# B&R Automation Studio project ChoiceBagging_SSBP
Automation Studio 4.5.2.102; Single Spout Bag Placer; technology packages: mapp 5.6.0

## Configuration SSBP1

CPU X20CP0410, AutomationRuntime D4.52, Build 4.1.2, Vc V4.52.0

### Hardware
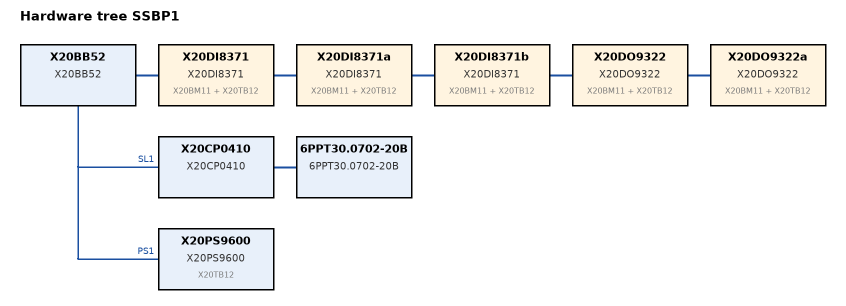
```
6PPT30.0702-20B : 6PPT30.0702-20B v1.1.0.0  [ETH1 -> X20CP0410.IF2 [Cable Type=PowerlinkCable, Length=10, Version=1.0.0.2]]
  Terminal = true
  PasswordVNC = 
  PasswordCIFS = 
  PasswordService = 
  VncKeyMappingFile = VC\6PPT30.0702-20B.dis
  VncRefreshRate = 400
X20BB52 : X20BB52 v1.1.0.0
X20BM11 : X20BM11 v1.0.0.1  [X2X1 -> X20BB52.IF6]
X20BM11a : X20BM11 v1.0.0.1  [X2X1 -> X20BM11d.X2X2]
X20BM11b : X20BM11 v1.0.0.1  [X2X1 -> X20BM11.X2X2]
X20BM11c : X20BM11 v1.0.0.1  [X2X1 -> X20BM11a.X2X2]
X20BM11d : X20BM11 v1.0.0.1  [X2X1 -> X20BM11b.X2X2]
X20CP0410 : X20CP0410 v1.2.1.0  [SL -> X20BB52.SL1]
  Connector IF2:
    ActivateDevice = 1
    Mode = Manual
    InternetAddress = 10.128.131.200
    SubnetMask = 255.255.255.0
    InaNodeNumber = 0
    Vnc1
    VncVcObjectName1 = Visu
    VncKeyMappingFile1 = VC\PS2-Keyboard.dis
    VncRefreshRate1 = 250
  ConfigurationID = ChoiceBagging_SSBP_SSBP1
  EnableUsbRemoteInstall = 1
  TimerDeviceType = SWIOTIMER
  Cyclic1Duration = 10000
  Cyclic1Tolerance = 10000
  Cyclic1Output = 1
  Cyclic2Duration = 20000
  Cyclic2Tolerance = 20000
  Cyclic3Duration = 50000
  Cyclic3Tolerance = 50000
  Cyclic4Duration = 100000
  Cyclic4Tolerance = 100000
  Cyclic5Duration = 200000
  Cyclic5Tolerance = 200000
  Cyclic6Duration = 500000
  Cyclic6Tolerance = 500000
  Cyclic7Duration = 1000000
  Cyclic7Tolerance = 1000000
  Cyclic8Duration = 10000
  Cyclic8Tolerance = 30000000
  ActivateOpcUa = 1
  OpcUaInformationModels_PV_Version = 1
X20DI8371 : X20DI8371 v1.0.2.0  [SS1 -> X20TB12a.SS; SL -> X20BM11.SL1]
  Supervision = off
X20DI8371a : X20DI8371 v1.0.2.0  [SS1 -> X20TB12c.SS; SL -> X20BM11b.SL1]
  Supervision = off
X20DI8371b : X20DI8371 v1.0.2.0  [SS1 -> X20TB12e.SS; SL -> X20BM11d.SL1]
X20DO9322 : X20DO9322 v1.0.3.0  [SS1 -> X20TB12b.SS; SL -> X20BM11a.SL1]
  Supervision = off
X20DO9322a : X20DO9322 v1.0.3.0  [SS1 -> X20TB12d.SS; SL -> X20BM11c.SL1]
  Supervision = off
X20PS9600 : X20PS9600 v1.0.1.0  [PS -> X20BB52.PS1; SS1 -> X20TB12.SS]
  Supervision = off
X20TB12 : X20TB12 v1.0.0.0
X20TB12a : X20TB12 v1.0.0.0
X20TB12b : X20TB12 v1.0.0.0
X20TB12c : X20TB12 v1.0.0.0
X20TB12d : X20TB12 v1.0.0.0
X20TB12e : X20TB12 v1.0.0.0
```

### IoMap.iom - X20CP0410/IoMap.iom
```iecst
VAR_CONFIG
	::gModuleOK.PowerSupply AT %IX."X20PS9600".ModuleOk;
	::gModuleOK.DigitalInput AT %IX."X20DI8371".ModuleOk;
	::gModuleOK.DigitalOutput AT %IX."X20DO9322".ModuleOk;
	::gModuleOK.DigitalInputa AT %IX."X20DI8371a".ModuleOk;
	::gModuleOK.DigitalOutputa AT %IX."X20DO9322a".ModuleOk;
	::gdi.L1CarriageRight AT %IX."X20DI8371".DigitalInput01;
	::gdi.L2CarriageLeft AT %IX."X20DI8371".DigitalInput02;
	::gdi.L3BagLifterUpper AT %IX."X20DI8371".DigitalInput03;
	::gdi.L4BagLifterLower AT %IX."X20DI8371".DigitalInput04;
	::gdi.L5DuckBillLeft AT %IX."X20DI8371".DigitalInput05;
	::gdi.L6DuckBillRight AT %IX."X20DI8371".DigitalInput06;
	::gdi.L7GripperOpen AT %IX."X20DI8371".DigitalInput07;
	::gdi.L8VacuumConfirm AT %IX."X20DI8371".DigitalInput08;
	::gdi.L9SwingArmUpper AT %IX."X20DI8371a".DigitalInput01;
	::gdi.L10SwingArmLower AT %IX."X20DI8371a".DigitalInput02;
	::gdi.L11EmptyBagInboundConv AT %IX."X20DI8371a".DigitalInput03;
	::gdi.L12Cyl7SpreaderSwitch AT %IX."X20DI8371a".DigitalInput04;
	::gdi.Bagger1Ready AT %IX."X20DI8371a".DigitalInput05;
	::gdi.Bagger2OnSpout AT %IX."X20DI8371a".DigitalInput06;
	::gdi.ConveyorOn AT %IX."X20DI8371a".DigitalInput07;
	::gdo.Cyl1CarriageLeft AT %QX."X20DO9322".DigitalOutput01;
	::gdo.Cyl1CarriageRight AT %QX."X20DO9322".DigitalOutput02;
	::gdo.Cyl2SwingArmUp AT %QX."X20DO9322".DigitalOutput03;
	::gdo.Cyl2SwingArmDown AT %QX."X20DO9322".DigitalOutput04;
	::gdo.Cyl3EmptyBagUp AT %QX."X20DO9322".DigitalOutput05;
	::gdo.Cyl3DownToEmptyBag AT %QX."X20DO9322".DigitalOutput06;
	::gdo.Cyl4DuckBillLeft AT %QX."X20DO9322".DigitalOutput07;
	::gdo.Cyl4DuckBillRight AT %QX."X20DO9322".DigitalOutput08;
	::gdo.Cyl5DuckBillIn AT %QX."X20DO9322".DigitalOutput09;
	::gdo.Cyl5DuckBillOut AT %QX."X20DO9322".DigitalOutput10;
	::gdo.Cyl6DuckBillOpen AT %QX."X20DO9322".DigitalOutput11;
	::gdo.Cyl6DuckBillClose AT %QX."X20DO9322".DigitalOutput12;
	::gdo.Cyl7Spreader AT %QX."X20DO9322a".DigitalOutput01;
	::gdo.Cyl8DropOpen AT %QX."X20DO9322a".DigitalOutput02;
	::gdo.Cyl8GripClose AT %QX."X20DO9322a".DigitalOutput03;
	::gdo.Vac1 AT %QX."X20DO9322a".DigitalOutput04;
	::gdo.Purge1 AT %QX."X20DO9322a".DigitalOutput05;
	::gdi.SafeToRun AT %IX."X20DI8371a".DigitalInput08;
	::gdi.ChairDischarge AT %IX."X20DI8371b".DigitalInput01;
	::gModuleOK.DigitalInputb AT %IX."X20DI8371b".ModuleOk;
	::gdo.Alarm AT %QX."X20DO9322a".DigitalOutput06;
	::gdo.Running AT %QX."X20DO9322a".DigitalOutput07;
	::gdi.SealerArmUp AT %IX."X20DI8371b".DigitalInput02;
	::gdi.ChairIn AT %IX."X20DI8371b".DigitalInput03;
END_VAR
```

### Config.mpalarmxcore - X20CP0410/mappServices/Config.mpalarmxcore
```
Element gAlarmXCore (Type=mpalarmxcore)
  mapp.AlarmX.Core.Configuration:
    [0]:
      Name = HomingTimeout
      Message = Timeout while homing machine.
      Code = 1
    [1]:
      Name = SafetyStatus
      Message = Safety status error not OK.
      Code = 2
    [2]:
      Name = ConveyorStatus
      Message = Conveyor status error not OK.
      Code = 3
    [3]:
      Name = ModuleStatus
      Message = Hardware module not OK.
      Code = 4
    [4]:
      Name = VacuumFailure
      Message = Vacuum confirmation failure.
      Code = 5
    [5]:
      Name = Bagger2Failure
      Message = No bag on spout.
      Code = 6
```

## Logical view

Binary libraries used (declarations not repeated): operator, runtime, astime, AsIecCon, AsArSdm, brsystem, MpBase, standard, sys_lib, MpAlarmX 5.06.0

### Global.typ - Global data types
```iecst
TYPE
	MachineState_type : 	STRUCT  (*State machine*)
		Sub0 : BOOL; (*Subroutine 0*)
		Sub1 : BOOL; (*Subroutine 1*)
		Sub2 : BOOL; (*Subroutine 2*)
		Sub3 : BOOL; (*Subroutine 3*)
		Sub4 : BOOL; (*Subroutine 4*)
		Sub5 : BOOL; (*Subroutine 5*)
		Sub6 : BOOL; (*Subroutine 6*)
		Sub7 : BOOL; (*Subroutine 7*)
		Sub8 : BOOL; (*Subroutine 8*)
		Sub9 : BOOL; (*Subroutine 9*)
	END_STRUCT;
	di_type : 	STRUCT  (*Digital inputs*)
		L1CarriageRight : BOOL; (*Carriage limit right*)
		L2CarriageLeft : BOOL; (*Carriage limit left*)
		L3BagLifterUpper : BOOL; (*Bag lifter limit upper*)
		L4BagLifterLower : BOOL; (*Bag lifter limit lower*)
		L5DuckBillLeft : BOOL; (*Duck bill limit left*)
		L6DuckBillRight : BOOL; (*Duck bill limit right*)
		L7GripperOpen : BOOL; (*Gripper open limit*)
		L8VacuumConfirm : BOOL; (*Vacuum confirmation*)
		L9SwingArmUpper : BOOL; (*Swing arm limit upper*)
		L10SwingArmLower : BOOL; (*Swing arm limit lower*)
		L11EmptyBagInboundConv : BOOL; (*Empty bag inbound conveyor*)
		L12Cyl7SpreaderSwitch : BOOL; (*Activate Cyl7 switch*)
		Bagger1Ready : BOOL; (*Ready signal from bagger*)
		Bagger2OnSpout : BOOL; (*No bag on spout from bagger*)
		ConveyorOn : BOOL; (*Conveyor on signal from robotic palletizer*)
		SafeToRun : BOOL; (*Safe to run signal from safety light curtain*)
		ChairDischarge : BOOL; (*Chair discharge signal*)
		SealerArmUp : BOOL; (*Sealer arm up signal*)
		ChairIn : BOOL; (*Chair in signal*)
	END_STRUCT;
	do_type : 	STRUCT  (*Digital outputs*)
		Cyl1CarriageLeft : BOOL; (*Move carriage left*)
		Cyl1CarriageRight : BOOL; (*Move carriage right*)
		Cyl2SwingArmUp : BOOL; (*Move swinging arm up*)
		Cyl2SwingArmDown : BOOL; (*Move swinging arm down*)
		Cyl3EmptyBagUp : BOOL; (*Lift empty bags up*)
		Cyl3DownToEmptyBag : BOOL; (*Move down to empty bags*)
		Cyl4DuckBillLeft : BOOL; (*Move duck bill assembly left*)
		Cyl4DuckBillRight : BOOL; (*Move duck bill assembly right*)
		Cyl5DuckBillIn : BOOL; (*Move duck bill in*)
		Cyl5DuckBillOut : BOOL; (*Move duck bill out*)
		Cyl6DuckBillOpen : BOOL; (*Open duck bill*)
		Cyl6DuckBillClose : BOOL; (*Close duck bill*)
		Cyl7Spreader : BOOL; (*Bag valve spreader*)
		Cyl8DropOpen : BOOL; (*Drop bag*)
		Cyl8GripClose : BOOL; (*Grip bag*)
		Vac1 : BOOL; (*Attach bag to bag lifter*)
		Purge1 : BOOL; (*Purge vacuum lines*)
		Alarm : BOOL; (*Error present*)
		Running : BOOL; (*Machine running*)
	END_STRUCT;
	ModuleOK_type : 	STRUCT  (*Module statuses*)
		PowerSupply : BOOL; (*X20PS9600 status*)
		DigitalInput : BOOL; (*X20DI8371 status*)
		DigitalOutput : BOOL; (*X20DO9322 status*)
		DigitalInputa : BOOL; (*X20DI8371a status*)
		DigitalOutputa : BOOL; (*X20DO9322a status*)
		DigitalInputb : BOOL; (*X20DI8371b status*)
	END_STRUCT;
	Timer_type : 	STRUCT  (*System timers*)
		HomePos : TIME; (*Homing Position timer value*)
		BagOnSpout : TIME; (*Bag on Spout timer value*)
		VacuumConfirm : TIME; (*Vacuum Confirmation timer value*)
		Cyl5 : TIME; (*Cyl 5 timer value*)
		Cyl6 : TIME; (*Cyl 6 timer value*)
		Cyl7 : TIME; (*Cyl 7 timer value*)
		GripperRetract : TIME; (*Gripper retract timer value*)
		SwingArm : TIME; (*Swing arm timer value*)
	END_STRUCT;
	Machine_type : 	STRUCT  (*Machine structure type*)
		Cmd : MachineCmd_type; (*Machine commands*)
		Par : MachinePar_type; (*Machine parameters*)
		Sts : MachineSts_type; (*Machine statuses*)
	END_STRUCT;
	MachineCmd_type : 	STRUCT  (*Machine commands*)
		Home : BOOL; (*Home*)
		Initialize : BOOL; (*Initialize - start from home*)
		Start : BOOL; (*Start machine*)
		Stop : BOOL; (*Stop machine*)
		ErrorReset : BOOL; (*Reset error*)
		Wait : BOOL; (*Wait state*)
		Pause : BOOL; (*Pause machine*)
		Resume : BOOL; (*Resume subroutine*)
	END_STRUCT;
	MachinePar_type : 	STRUCT  (*Machine parameters*)
		VacuumFail : UDINT; (*Vacuum confirmation failure*)
		VacuumFailTotal : UDINT; (*Vacuum confirmation failure total*)
		Bagger2Fail : UDINT; (*Bagger 2 on Spout failure*)
		Bagger2FailTotal : UDINT; (*Bagger 2 on Spout failure total*)
	END_STRUCT;
	MachineSts_type : 	STRUCT  (*Machine statuses*)
		IsHomed : BOOL; (*Is homed*)
		Cyl6LimitClose : BOOL; (*Cyl 6 timer feedback - duck bill close*)
		Cyl6LimitOpen : BOOL; (*Cyl 6 timer feedback - duck bill open*)
		Cyl5LimitOut : BOOL; (*Cyl 5 timer feedback - duck bill out*)
		Cyl5LimitIn : BOOL; (*Cyl 5 timer feedback - duck bill in*)
		Error : BOOL; (*Error detected*)
		HomePosTimeout : BOOL; (*Home Position timeout*)
		VacuumTimeout : BOOL; (*Vacuum Confirmation timeout*)
		AttemptsLeft : BOOL; (*Attempts left before error - vacuum*)
		NoAttemptsLeft : BOOL; (*No vacuum attempts left - error*)
		Bagger2Timeout : BOOL; (*Bag on Spout timeout*)
		BaggerAttemptsLeft : BOOL; (*Attempts left before error - Bagger 2*)
		NoBaggerAttemptsLeft : BOOL; (*No Bagger 2 attempts left - error*)
	END_STRUCT;
	Input_type : 	STRUCT  (*Machine inputs*)
		L1CarriageRight : BOOL; (*Carriage limit right*)
		L2CarriageLeft : BOOL; (*Carriage limit left*)
		L3BagLifterUpper : BOOL; (*Bag lifter limit upper*)
		L4BagLifterLower : BOOL; (*Bag lifter limit lower*)
		L5DuckBillLeft : BOOL; (*Duck bill limit left*)
		L6DuckBillRight : BOOL; (*Duck bill limit right*)
		L7GripperOpen : BOOL; (*Gripper open limit*)
		L8VacuumConfirm : BOOL; (*Vacuum confirmation*)
		L9SwingArmUpper : BOOL; (*Swing arm limit upper*)
		L10SwingArmLower : BOOL; (*Swing arm limit lower*)
		L11EmptyBagInboundConv : BOOL; (*Empty bag inbound conveyor*)
		L12Cyl7SpreaderSwitch : BOOL; (*Activate Cyl7 switch*)
		Bagger1Ready : BOOL; (*Ready signal from bagger*)
		Bagger2OnSpout : BOOL; (*No bag on spout from bagger*)
		ConveyorOn : BOOL; (*Conveyor on signal from robotic palletizer*)
		SafeToRun : BOOL; (*Safe to run signal from safety light curtain*)
		ChairDischarge : BOOL; (*Chair discharge signal*)
		SealerArmUp : BOOL; (*Sealer arm up signal*)
		ChairIn : BOOL; (*Chair in signal*)
	END_STRUCT;
	Output_type : 	STRUCT  (*Machine outputs*)
		Cyl1CarriageLeft : BOOL; (*Move carriage left*)
		Cyl1CarriageRight : BOOL; (*Move carriage right*)
		Cyl2SwingArmUp : BOOL; (*Move swinging arm up*)
		Cyl2SwingArmDown : BOOL; (*Move swinging arm down*)
		Cyl3EmptyBagUp : BOOL; (*Lift empty bags up*)
		Cyl3DownToEmptyBag : BOOL; (*Move down to empty bags*)
		Cyl4DuckBillLeft : BOOL; (*Move duck bill assembly left*)
		Cyl4DuckBillRight : BOOL; (*Move duck bill assembly right*)
		Cyl5DuckBillIn : BOOL; (*Move duck bill in*)
		Cyl5DuckBillOut : BOOL; (*Move duck bill out*)
		Cyl6DuckBillOpen : BOOL; (*Open duck bill*)
		Cyl6DuckBillClose : BOOL; (*Close duck bill*)
		Cyl7Spreader : BOOL; (*Bag valve spreader*)
		Cyl8DropOpen : BOOL; (*Drop bag*)
		Cyl8GripClose : BOOL; (*Grip bag*)
		Vac1 : BOOL; (*Attach bag to bag lifter*)
		Purge1 : BOOL; (*Purge vacuum lines*)
		Alarm : BOOL; (*Error detected*)
		Running : BOOL; (*Machine Running*)
	END_STRUCT;
	ErrorID_enum :
		( (*Error ID enumeration*)
		HOMING_TIMEOUT := 1, (*Homing position timeout*)
		SAFE_TO_RUN := 2, (*Machine not Safe to Run*)
		CONVEYOR := 3, (*Conveyor not on*)
		MODULE_OK := 4, (*Module OK status error*)
		VACUUM_FAILURE := 5, (*Vacuum failure (after 3 attempts)*)
		BAG_ON_SPOUT_FAILURE := 6 (*No Bag on spout (after 3 attempts)*)
		);
END_TYPE
```

### Global.var - Global variables
```iecst
VAR
	gdi : di_type; (*Digital inputs*)
	gdo : do_type; (*Digital outputs*)
	gModuleOK : ModuleOK_type; (*Module statuses*)
	gTimer : Timer_type; (*System timers*)
	gErrorID : UDINT; (*Error ID*)
	gMachine : Machine_type; (*Machine process variable*)
	gInput : Input_type; (*Machine inputs process variable*)
	gOutput : Output_type; (*Machine outputs process variable*)
	gMachineState : MachineState_type; (*State machine process variable*)
END_VAR
```


### Program Logical/MainCtrl (IEC)

#### Cyclic.ld - Cyclic code
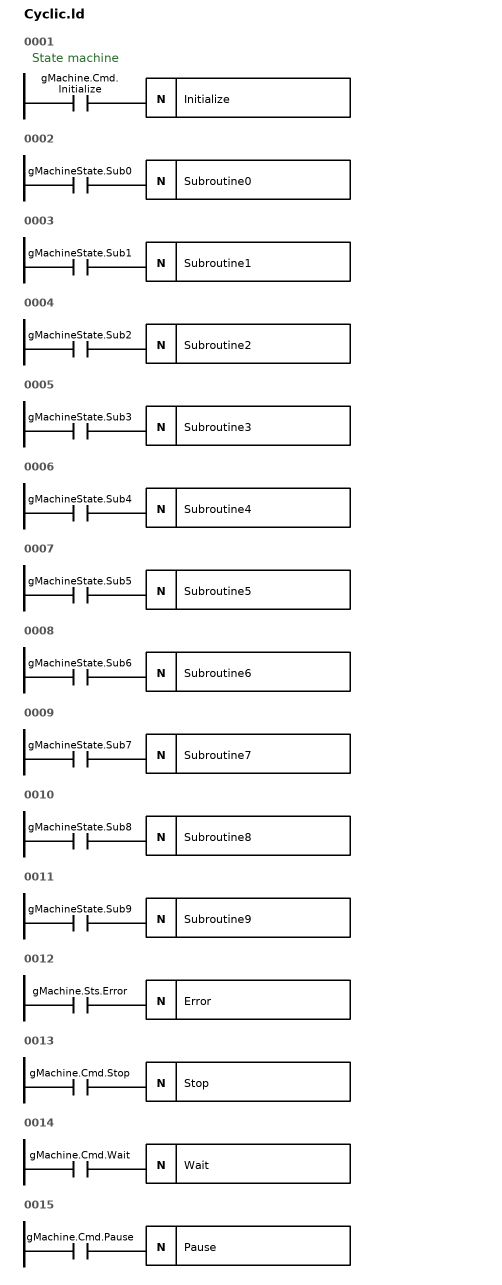
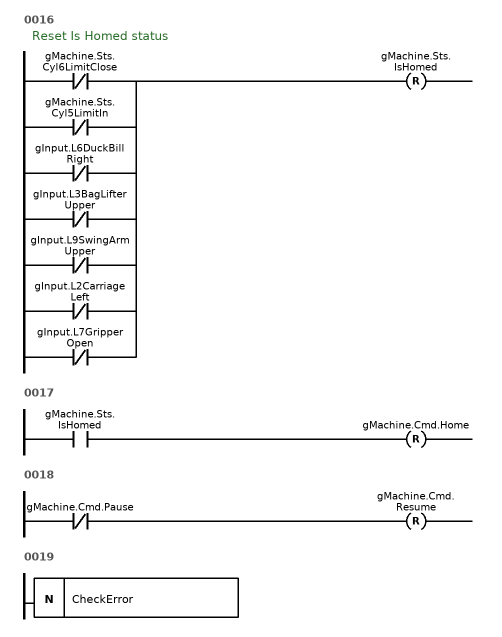
Ladder, written as Structured Text:
```iecst
(*********************************************************************************
 * Copyright: 	Hartfiel Automation
 * Author:    	cashley
 * Created:   	August 5, 2019/2:01 PM
 * Description: This file contains the main control logic for the machine.
 *********************************************************************************)
 PROGRAM _CYCLIC
(* Network 1: State machine *)
IF gMachine.Cmd.Initialize THEN Initialize; END_IF;

(* Network 2 *)
IF gMachineState.Sub0 THEN Subroutine0; END_IF;

(* Network 3 *)
IF gMachineState.Sub1 THEN Subroutine1; END_IF;

(* Network 4 *)
IF gMachineState.Sub2 THEN Subroutine2; END_IF;

(* Network 5 *)
IF gMachineState.Sub3 THEN Subroutine3; END_IF;

(* Network 6 *)
IF gMachineState.Sub4 THEN Subroutine4; END_IF;

(* Network 7 *)
IF gMachineState.Sub5 THEN Subroutine5; END_IF;

(* Network 8 *)
IF gMachineState.Sub6 THEN Subroutine6; END_IF;

(* Network 9 *)
IF gMachineState.Sub7 THEN Subroutine7; END_IF;

(* Network 10 *)
IF gMachineState.Sub8 THEN Subroutine8; END_IF;

(* Network 11 *)
IF gMachineState.Sub9 THEN Subroutine9; END_IF;

(* Network 12 *)
IF gMachine.Sts.Error THEN Error; END_IF;

(* Network 13 *)
IF gMachine.Cmd.Stop THEN Stop; END_IF;

(* Network 14 *)
IF gMachine.Cmd.Wait THEN Wait; END_IF;

(* Network 15 *)
IF gMachine.Cmd.Pause THEN Pause; END_IF;

(* Network 16: Reset Is Homed status *)
IF NOT gMachine.Sts.Cyl6LimitClose OR NOT gMachine.Sts.Cyl5LimitIn OR NOT gInput.L6DuckBillRight OR NOT gInput.L3BagLifterUpper OR NOT gInput.L9SwingArmUpper OR NOT gInput.L2CarriageLeft OR NOT gInput.L7GripperOpen THEN
    gMachine.Sts.IsHomed := FALSE;
END_IF;

(* Network 17 *)
IF gMachine.Sts.IsHomed THEN gMachine.Cmd.Home := FALSE; END_IF;

(* Network 18 *)
IF NOT gMachine.Cmd.Pause THEN gMachine.Cmd.Resume := FALSE; END_IF;

(* Network 19 *)
CheckError;
END_PROGRAM
```

#### Init.ld - Initialization code
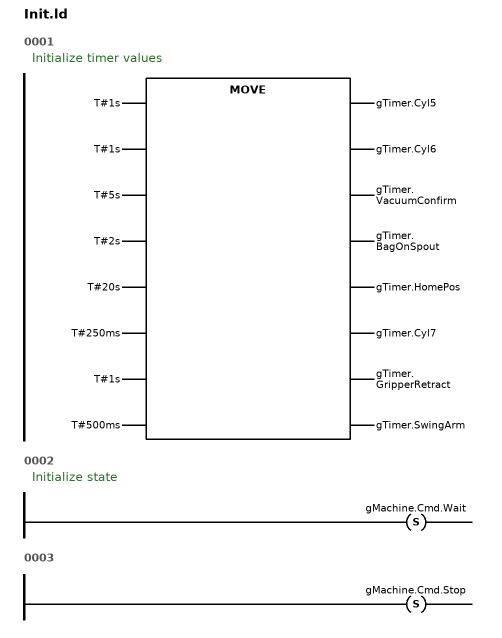
Ladder, written as Structured Text:
```iecst
PROGRAM _INIT
(* Network 1: Initialize timer values *)
gTimer.Cyl5 := T#1s;
gTimer.Cyl6 := T#1s;
gTimer.VacuumConfirm := T#5s;
gTimer.BagOnSpout := T#2s;
gTimer.HomePos := T#20s;
gTimer.Cyl7 := T#250ms;
gTimer.GripperRetract := T#1s;
gTimer.SwingArm := T#500ms;

(* Network 2: Initialize state *)
gMachine.Cmd.Wait := TRUE;

(* Network 3 *)
gMachine.Cmd.Stop := TRUE;
END_PROGRAM
```

#### Variables.var - Local variables
```iecst
VAR
	TON_Cyl6 : TON; (*TON function block for Cyl 6 timer*)
	TON_Cyl5 : TON; (*TON function block for Cyl 5 timer*)
	TON_VacuumConfirm : TON; (*TON function block for Vacuum Confirmation timer*)
	TON_BagOnSpout : TON; (*TON function block for Bag on Spout timer*)
	TON_HomePos : TON; (*TON function block for Homing Position timer*)
	TON_Cyl7Switch : TON; (*TON function block for Cyl 7 Spreader Switch timer*)
END_VAR
VAR CONSTANT
	Cyl7SwitchTimer : TIME := T#3S; (*Cyl7 Spreader Switch timer value*)
END_VAR
VAR
	TON_Cyl3 : TON; (*TON function block for Cyl3 timer*)
	ExecuteJump : BOOL; (*Jump to repeat three times before error*)
	TON_Cyl5_Sub2 : TON; (*TON function block for Cyl 5 timer in Subroutine 2*)
	TON_Cyl6_Sub2 : TON; (*TON function block for Cyl 6 timer in Subroutine 2*)
	TON_Cyl5_Sub0 : TON; (*TON function block for Cyl 5 timer in Subroutine 0*)
	TON_Cyl6_Sub0 : TON; (*TON function block for Cyl 6 timer in Subroutine 0*)
	TON_Cyl5_Sub4 : TON; (*TON function block for Cyl 5 timer in Subroutine 4*)
	TON_Cyl6_Sub4 : TON; (*TON function block for Cyl 6 timer in Subroutine 4*)
	TON_Cyl6_Sub4_2 : TON; (*TON function block for Cyl 6 timer #2 in Subroutine 4*)
	TON_GripperRetract : TON; (*TON function block for Gripper Retract timer*)
	TON_SwingArm : TON; (*TON function block for Swing Arm timer*)
	StateOld : UDINT; (*Last machine state*)
	StateOldIsSet : BOOL; (*Last machine state is set*)
END_VAR
```

#### Initialize.ld - Start from home
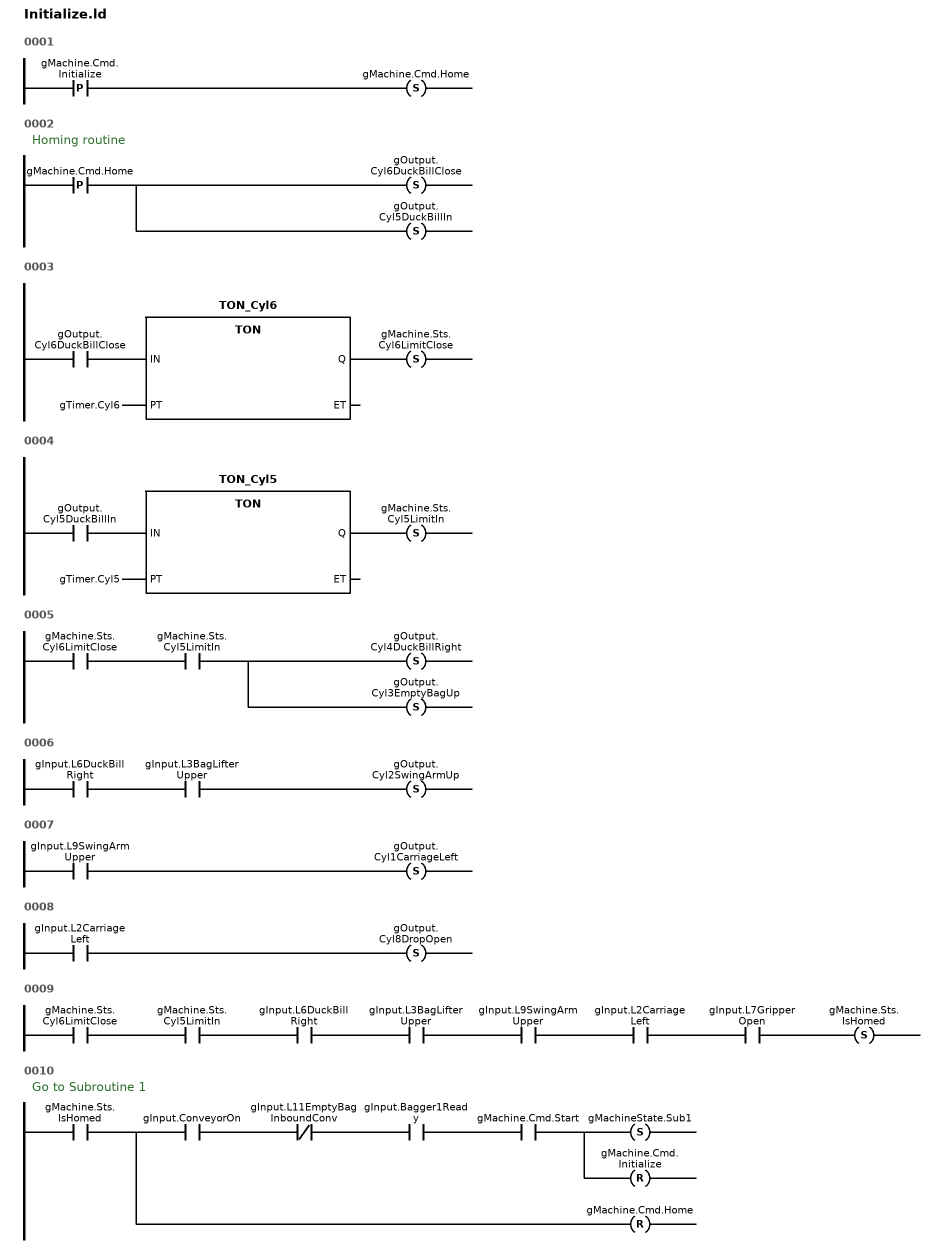
Ladder, written as Structured Text:
```iecst
ACTION Initialize:
VAR
    _e1 : R_TRIG;
    _e2 : R_TRIG;
    _p3 : BOOL;
    _p4 : BOOL;
    _p5 : BOOL;
END_VAR
(* Network 1 *)
_e1(CLK := gMachine.Cmd.Initialize);
IF _e1.Q THEN gMachine.Cmd.Home := TRUE; END_IF;

(* Network 2: Homing routine *)
_e2(CLK := gMachine.Cmd.Home);
IF _e2.Q THEN
    gOutput.Cyl6DuckBillClose := TRUE;
    gOutput.Cyl5DuckBillIn := TRUE;
END_IF;

(* Network 3 *)
TON_Cyl6(IN := gOutput.Cyl6DuckBillClose, PT := gTimer.Cyl6);
IF TON_Cyl6.Q THEN gMachine.Sts.Cyl6LimitClose := TRUE; END_IF;

(* Network 4 *)
TON_Cyl5(IN := gOutput.Cyl5DuckBillIn, PT := gTimer.Cyl5);
IF TON_Cyl5.Q THEN gMachine.Sts.Cyl5LimitIn := TRUE; END_IF;

(* Network 5 *)
_p3 := gMachine.Sts.Cyl6LimitClose AND gMachine.Sts.Cyl5LimitIn;
IF _p3 THEN
    gOutput.Cyl4DuckBillRight := TRUE;
    gOutput.Cyl3EmptyBagUp := TRUE;
END_IF;

(* Network 6 *)
IF gInput.L6DuckBillRight AND gInput.L3BagLifterUpper THEN gOutput.Cyl2SwingArmUp := TRUE; END_IF;

(* Network 7 *)
IF gInput.L9SwingArmUpper THEN gOutput.Cyl1CarriageLeft := TRUE; END_IF;

(* Network 8 *)
IF gInput.L2CarriageLeft THEN gOutput.Cyl8DropOpen := TRUE; END_IF;

(* Network 9 *)
IF gMachine.Sts.Cyl6LimitClose AND gMachine.Sts.Cyl5LimitIn AND gInput.L6DuckBillRight AND gInput.L3BagLifterUpper AND gInput.L9SwingArmUpper AND gInput.L2CarriageLeft AND gInput.L7GripperOpen THEN
    gMachine.Sts.IsHomed := TRUE;
END_IF;

(* Network 10: Go to Subroutine 1 *)
_p4 := gMachine.Sts.IsHomed AND gInput.ConveyorOn AND NOT gInput.L11EmptyBagInboundConv AND gInput.Bagger1Ready AND gMachine.Cmd.Start;
IF _p4 THEN gMachineState.Sub1 := TRUE; END_IF;
_p5 := gMachine.Sts.IsHomed;
IF _p4 THEN gMachine.Cmd.Initialize := FALSE; END_IF;
IF _p5 THEN gMachine.Cmd.Home := FALSE; END_IF;
END_ACTION
```

#### Subroutine0.ld - Continuous running mode
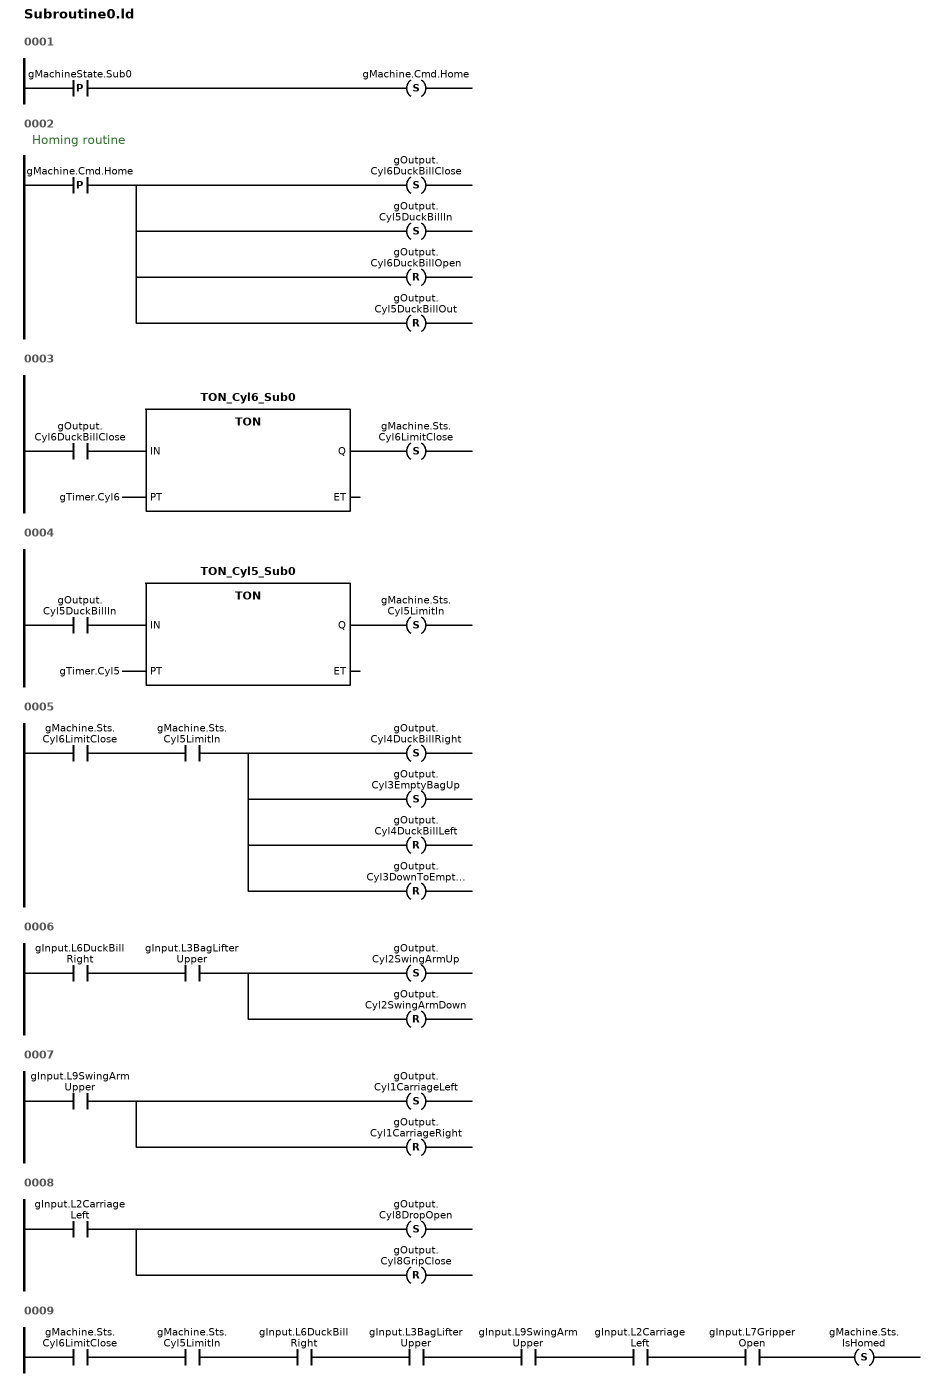
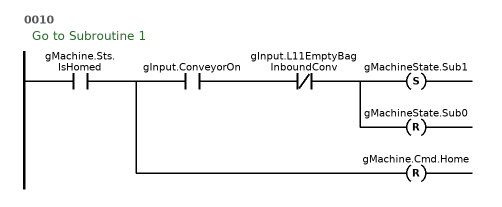
Ladder, written as Structured Text:
```iecst
ACTION Subroutine0:
VAR
    _e1 : R_TRIG;
    _e2 : R_TRIG;
    _p3 : BOOL;
    _p4 : BOOL;
    _p5 : BOOL;
END_VAR
(* Network 1 *)
_e1(CLK := gMachineState.Sub0);
IF _e1.Q THEN gMachine.Cmd.Home := TRUE; END_IF;

(* Network 2: Homing routine *)
_e2(CLK := gMachine.Cmd.Home);
IF _e2.Q THEN
    gOutput.Cyl6DuckBillClose := TRUE;
    gOutput.Cyl5DuckBillIn := TRUE;
    gOutput.Cyl6DuckBillOpen := FALSE;
    gOutput.Cyl5DuckBillOut := FALSE;
END_IF;

(* Network 3 *)
TON_Cyl6_Sub0(IN := gOutput.Cyl6DuckBillClose, PT := gTimer.Cyl6);
IF TON_Cyl6_Sub0.Q THEN gMachine.Sts.Cyl6LimitClose := TRUE; END_IF;

(* Network 4 *)
TON_Cyl5_Sub0(IN := gOutput.Cyl5DuckBillIn, PT := gTimer.Cyl5);
IF TON_Cyl5_Sub0.Q THEN gMachine.Sts.Cyl5LimitIn := TRUE; END_IF;

(* Network 5 *)
_p3 := gMachine.Sts.Cyl6LimitClose AND gMachine.Sts.Cyl5LimitIn;
IF _p3 THEN
    gOutput.Cyl4DuckBillRight := TRUE;
    gOutput.Cyl3EmptyBagUp := TRUE;
    gOutput.Cyl4DuckBillLeft := FALSE;
    gOutput.Cyl3DownToEmptyBag := FALSE;
END_IF;

(* Network 6 *)
_p4 := gInput.L6DuckBillRight AND gInput.L3BagLifterUpper;
IF _p4 THEN
    gOutput.Cyl2SwingArmUp := TRUE;
    gOutput.Cyl2SwingArmDown := FALSE;
END_IF;

(* Network 7 *)
IF gInput.L9SwingArmUpper THEN
    gOutput.Cyl1CarriageLeft := TRUE;
    gOutput.Cyl1CarriageRight := FALSE;
END_IF;

(* Network 8 *)
IF gInput.L2CarriageLeft THEN
    gOutput.Cyl8DropOpen := TRUE;
    gOutput.Cyl8GripClose := FALSE;
END_IF;

(* Network 9 *)
IF gMachine.Sts.Cyl6LimitClose AND gMachine.Sts.Cyl5LimitIn AND gInput.L6DuckBillRight AND gInput.L3BagLifterUpper AND gInput.L9SwingArmUpper AND gInput.L2CarriageLeft AND gInput.L7GripperOpen THEN
    gMachine.Sts.IsHomed := TRUE;
END_IF;

(* Network 10: Go to Subroutine 1 *)
_p5 := gMachine.Sts.IsHomed AND gInput.ConveyorOn AND NOT gInput.L11EmptyBagInboundConv;
IF _p5 THEN
    gMachineState.Sub1 := TRUE;
    gMachineState.Sub0 := FALSE;
END_IF;
IF gMachine.Sts.IsHomed THEN gMachine.Cmd.Home := FALSE; END_IF;
END_ACTION
```

#### Subroutine1.ld - Pick up / lift empty bags
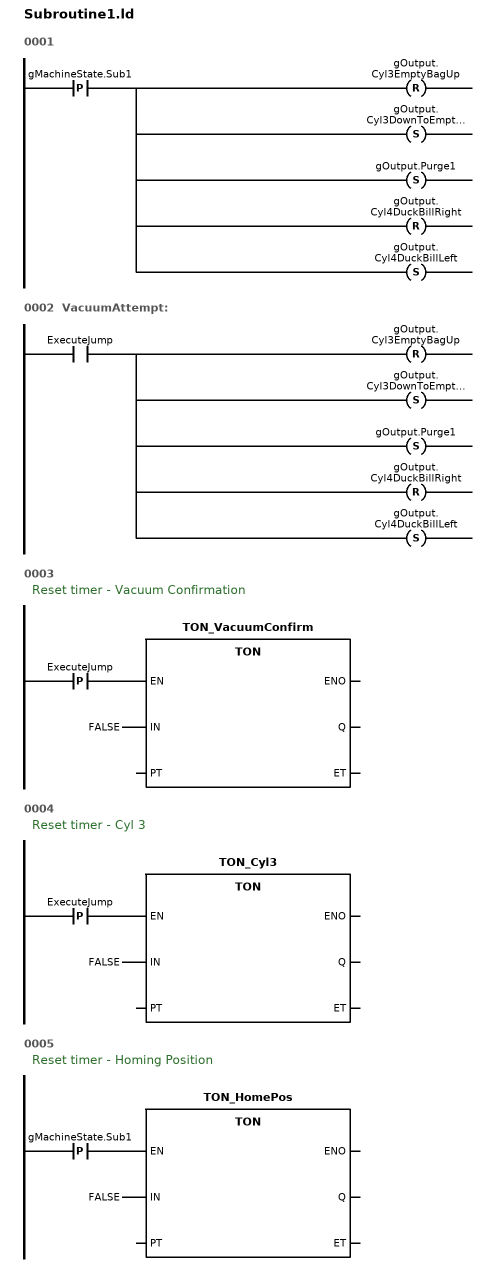
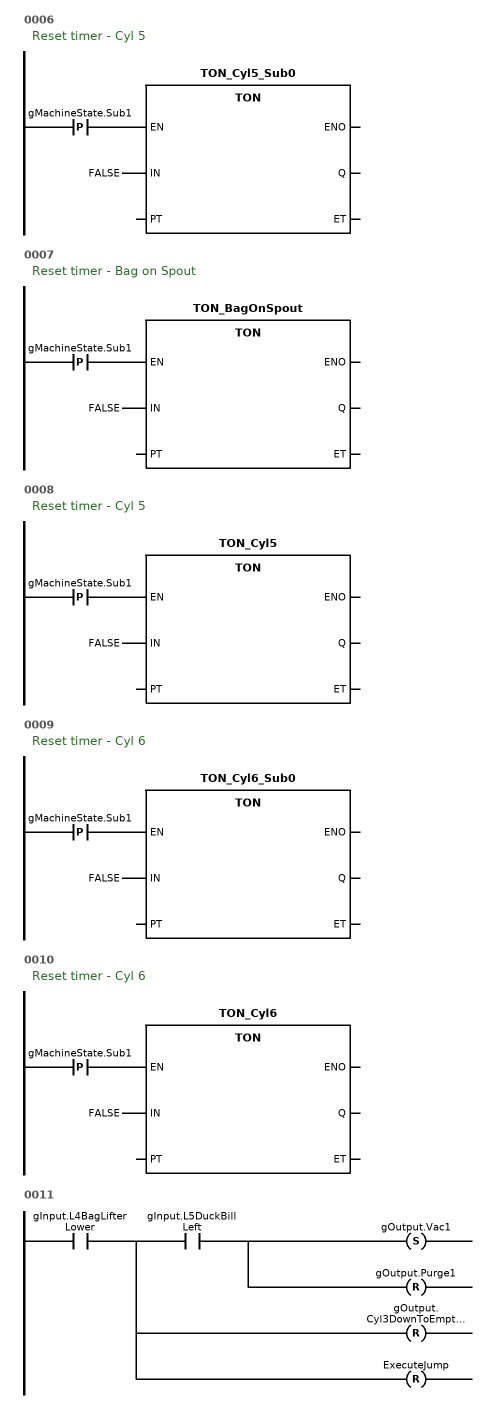
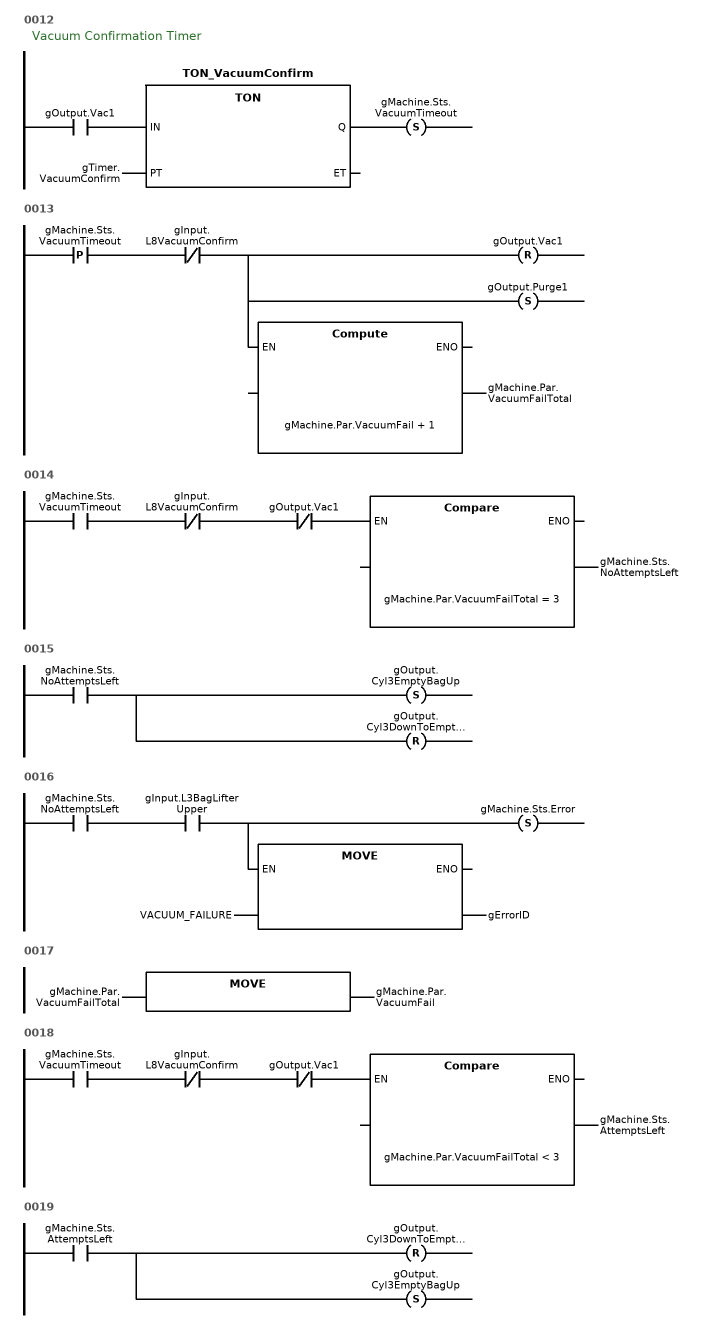
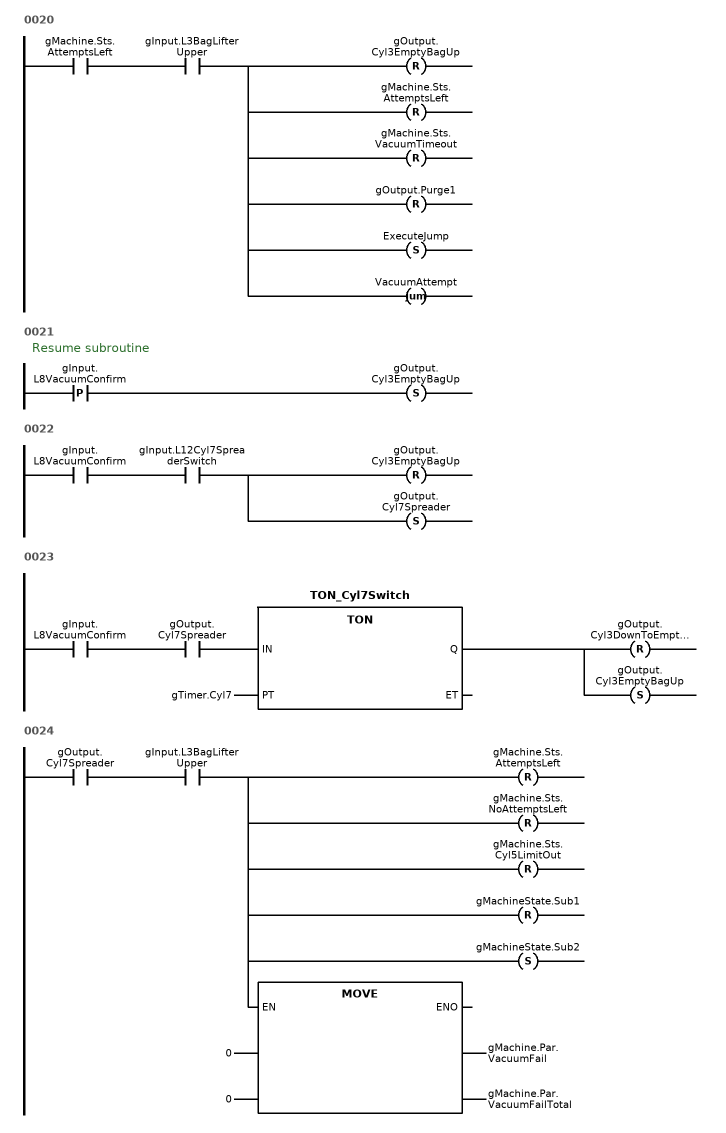
Ladder, written as Structured Text:
```iecst
ACTION Subroutine1:
VAR
    _e1 : R_TRIG;
    _e2 : R_TRIG;
    _e3 : R_TRIG;
    _e4 : R_TRIG;
    _e5 : R_TRIG;
    _e6 : R_TRIG;
    _e7 : R_TRIG;
    _e8 : R_TRIG;
    _e9 : R_TRIG;
    _p10 : BOOL;
    _e11 : R_TRIG;
    _p12 : BOOL;
    _p13 : BOOL;
    _p14 : BOOL;
    _p15 : BOOL;
    _e16 : R_TRIG;
    _p17 : BOOL;
END_VAR
(* Network 1 *)
_e1(CLK := gMachineState.Sub1);
IF _e1.Q THEN
    gOutput.Cyl3EmptyBagUp := FALSE;
    gOutput.Cyl3DownToEmptyBag := TRUE;
    gOutput.Purge1 := TRUE;
    gOutput.Cyl4DuckBillRight := FALSE;
    gOutput.Cyl4DuckBillLeft := TRUE;
END_IF;

(* Network 2 *)
VacuumAttempt:
IF ExecuteJump THEN
    gOutput.Cyl3EmptyBagUp := FALSE;
    gOutput.Cyl3DownToEmptyBag := TRUE;
    gOutput.Purge1 := TRUE;
    gOutput.Cyl4DuckBillRight := FALSE;
    gOutput.Cyl4DuckBillLeft := TRUE;
END_IF;

(* Network 3: Reset timer - Vacuum Confirmation *)
_e2(CLK := ExecuteJump);
IF _e2.Q THEN TON_VacuumConfirm(IN := FALSE); END_IF;

(* Network 4: Reset timer - Cyl 3 *)
_e3(CLK := ExecuteJump);
IF _e3.Q THEN TON_Cyl3(IN := FALSE); END_IF;

(* Network 5: Reset timer - Homing Position *)
_e4(CLK := gMachineState.Sub1);
IF _e4.Q THEN TON_HomePos(IN := FALSE); END_IF;

(* Network 6: Reset timer - Cyl 5 *)
_e5(CLK := gMachineState.Sub1);
IF _e5.Q THEN TON_Cyl5_Sub0(IN := FALSE); END_IF;

(* Network 7: Reset timer - Bag on Spout *)
_e6(CLK := gMachineState.Sub1);
IF _e6.Q THEN TON_BagOnSpout(IN := FALSE); END_IF;

(* Network 8: Reset timer - Cyl 5 *)
_e7(CLK := gMachineState.Sub1);
IF _e7.Q THEN TON_Cyl5(IN := FALSE); END_IF;

(* Network 9: Reset timer - Cyl 6 *)
_e8(CLK := gMachineState.Sub1);
IF _e8.Q THEN TON_Cyl6_Sub0(IN := FALSE); END_IF;

(* Network 10: Reset timer - Cyl 6 *)
_e9(CLK := gMachineState.Sub1);
IF _e9.Q THEN TON_Cyl6(IN := FALSE); END_IF;

(* Network 11 *)
_p10 := gInput.L4BagLifterLower AND gInput.L5DuckBillLeft;
IF _p10 THEN
    gOutput.Vac1 := TRUE;
    gOutput.Purge1 := FALSE;
END_IF;
IF gInput.L4BagLifterLower THEN
    gOutput.Cyl3DownToEmptyBag := FALSE;
    ExecuteJump := FALSE;
END_IF;

(* Network 12: Vacuum Confirmation Timer *)
TON_VacuumConfirm(IN := gOutput.Vac1, PT := gTimer.VacuumConfirm);
IF TON_VacuumConfirm.Q THEN gMachine.Sts.VacuumTimeout := TRUE; END_IF;

(* Network 13 *)
_e11(CLK := gMachine.Sts.VacuumTimeout);
IF _e11.Q AND NOT gInput.L8VacuumConfirm THEN
    gOutput.Vac1 := FALSE;
    gOutput.Purge1 := TRUE;
    gMachine.Par.VacuumFailTotal := gMachine.Par.VacuumFail + 1;
END_IF;

(* Network 14 *)
_p12 := gMachine.Sts.VacuumTimeout AND NOT gInput.L8VacuumConfirm AND NOT gOutput.Vac1;
IF _p12 THEN gMachine.Sts.NoAttemptsLeft := gMachine.Par.VacuumFailTotal = 3; END_IF;

(* Network 15 *)
IF gMachine.Sts.NoAttemptsLeft THEN
    gOutput.Cyl3EmptyBagUp := TRUE;
    gOutput.Cyl3DownToEmptyBag := FALSE;
END_IF;

(* Network 16 *)
_p13 := gMachine.Sts.NoAttemptsLeft AND gInput.L3BagLifterUpper;
IF _p13 THEN
    gMachine.Sts.Error := TRUE;
    gErrorID := VACUUM_FAILURE;
END_IF;

(* Network 17 *)
gMachine.Par.VacuumFail := gMachine.Par.VacuumFailTotal;

(* Network 18 *)
_p14 := gMachine.Sts.VacuumTimeout AND NOT gInput.L8VacuumConfirm AND NOT gOutput.Vac1;
IF _p14 THEN gMachine.Sts.AttemptsLeft := gMachine.Par.VacuumFailTotal < 3; END_IF;

(* Network 19 *)
IF gMachine.Sts.AttemptsLeft THEN
    gOutput.Cyl3DownToEmptyBag := FALSE;
    gOutput.Cyl3EmptyBagUp := TRUE;
END_IF;

(* Network 20 *)
_p15 := gMachine.Sts.AttemptsLeft AND gInput.L3BagLifterUpper;
IF _p15 THEN
    gOutput.Cyl3EmptyBagUp := FALSE;
    gMachine.Sts.AttemptsLeft := FALSE;
    gMachine.Sts.VacuumTimeout := FALSE;
    gOutput.Purge1 := FALSE;
    ExecuteJump := TRUE;
    JMP VacuumAttempt;
END_IF;

(* Network 21: Resume subroutine *)
_e16(CLK := gInput.L8VacuumConfirm);
IF _e16.Q THEN gOutput.Cyl3EmptyBagUp := TRUE; END_IF;

(* Network 22 *)
_p17 := gInput.L8VacuumConfirm AND gInput.L12Cyl7SpreaderSwitch;
IF _p17 THEN
    gOutput.Cyl3EmptyBagUp := FALSE;
    gOutput.Cyl7Spreader := TRUE;
END_IF;

(* Network 23 *)
TON_Cyl7Switch(IN := gInput.L8VacuumConfirm AND gOutput.Cyl7Spreader, PT := gTimer.Cyl7);
IF TON_Cyl7Switch.Q THEN
    gOutput.Cyl3DownToEmptyBag := FALSE;
    gOutput.Cyl3EmptyBagUp := TRUE;
END_IF;

(* Network 24 *)
IF gOutput.Cyl7Spreader AND gInput.L3BagLifterUpper THEN
    gMachine.Sts.AttemptsLeft := FALSE;
    gMachine.Sts.NoAttemptsLeft := FALSE;
    gMachine.Sts.Cyl5LimitOut := FALSE;
    gMachineState.Sub1 := FALSE;
    gMachineState.Sub2 := TRUE;
    gMachine.Par.VacuumFail := 0;
    gMachine.Par.VacuumFailTotal := 0;
END_IF;
END_ACTION
```

#### Subroutine2.ld - Insert duck bill / expand bill
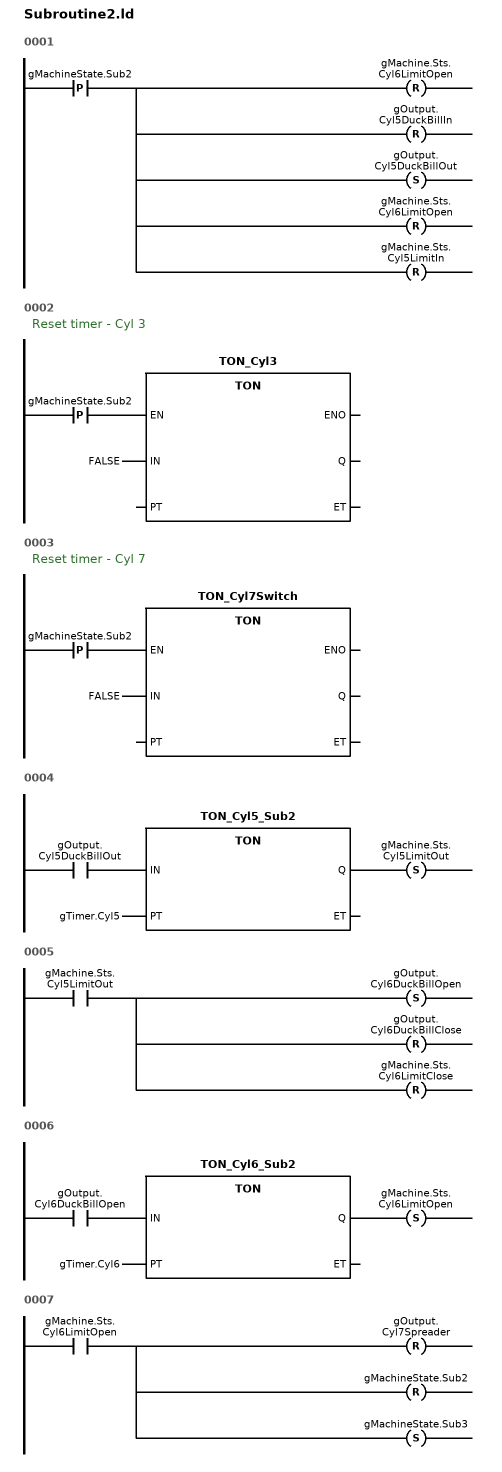
Ladder, written as Structured Text:
```iecst
ACTION Subroutine2:
VAR
    _e1 : R_TRIG;
    _e2 : R_TRIG;
    _e3 : R_TRIG;
END_VAR
(* Network 1 *)
_e1(CLK := gMachineState.Sub2);
IF _e1.Q THEN
    gMachine.Sts.Cyl6LimitOpen := FALSE;
    gOutput.Cyl5DuckBillIn := FALSE;
    gOutput.Cyl5DuckBillOut := TRUE;
    gMachine.Sts.Cyl6LimitOpen := FALSE;
    gMachine.Sts.Cyl5LimitIn := FALSE;
END_IF;

(* Network 2: Reset timer - Cyl 3 *)
_e2(CLK := gMachineState.Sub2);
IF _e2.Q THEN TON_Cyl3(IN := FALSE); END_IF;

(* Network 3: Reset timer - Cyl 7 *)
_e3(CLK := gMachineState.Sub2);
IF _e3.Q THEN TON_Cyl7Switch(IN := FALSE); END_IF;

(* Network 4 *)
TON_Cyl5_Sub2(IN := gOutput.Cyl5DuckBillOut, PT := gTimer.Cyl5);
IF TON_Cyl5_Sub2.Q THEN gMachine.Sts.Cyl5LimitOut := TRUE; END_IF;

(* Network 5 *)
IF gMachine.Sts.Cyl5LimitOut THEN
    gOutput.Cyl6DuckBillOpen := TRUE;
    gOutput.Cyl6DuckBillClose := FALSE;
    gMachine.Sts.Cyl6LimitClose := FALSE;
END_IF;

(* Network 6 *)
TON_Cyl6_Sub2(IN := gOutput.Cyl6DuckBillOpen, PT := gTimer.Cyl6);
IF TON_Cyl6_Sub2.Q THEN gMachine.Sts.Cyl6LimitOpen := TRUE; END_IF;

(* Network 7 *)
IF gMachine.Sts.Cyl6LimitOpen THEN
    gOutput.Cyl7Spreader := FALSE;
    gMachineState.Sub2 := FALSE;
    gMachineState.Sub3 := TRUE;
END_IF;
END_ACTION
```

#### Subroutine3.ld - Move bag to side
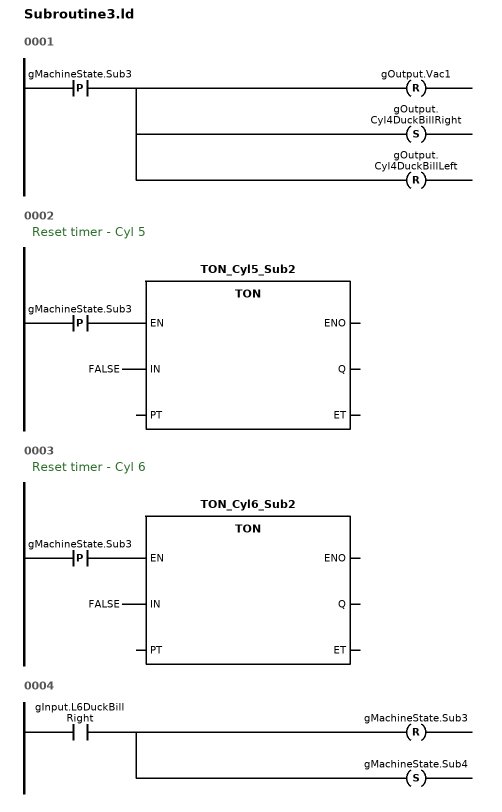
Ladder, written as Structured Text:
```iecst
ACTION Subroutine3:
VAR
    _e1 : R_TRIG;
    _e2 : R_TRIG;
    _e3 : R_TRIG;
END_VAR
(* Network 1 *)
_e1(CLK := gMachineState.Sub3);
IF _e1.Q THEN
    gOutput.Vac1 := FALSE;
    gOutput.Cyl4DuckBillRight := TRUE;
    gOutput.Cyl4DuckBillLeft := FALSE;
END_IF;

(* Network 2: Reset timer - Cyl 5 *)
_e2(CLK := gMachineState.Sub3);
IF _e2.Q THEN TON_Cyl5_Sub2(IN := FALSE); END_IF;

(* Network 3: Reset timer - Cyl 6 *)
_e3(CLK := gMachineState.Sub3);
IF _e3.Q THEN TON_Cyl6_Sub2(IN := FALSE); END_IF;

(* Network 4 *)
IF gInput.L6DuckBillRight THEN
    gMachineState.Sub3 := FALSE;
    gMachineState.Sub4 := TRUE;
END_IF;
END_ACTION
```

#### Subroutine4.ld - Swing bag gripper over duck bill / grab bag / shut bill
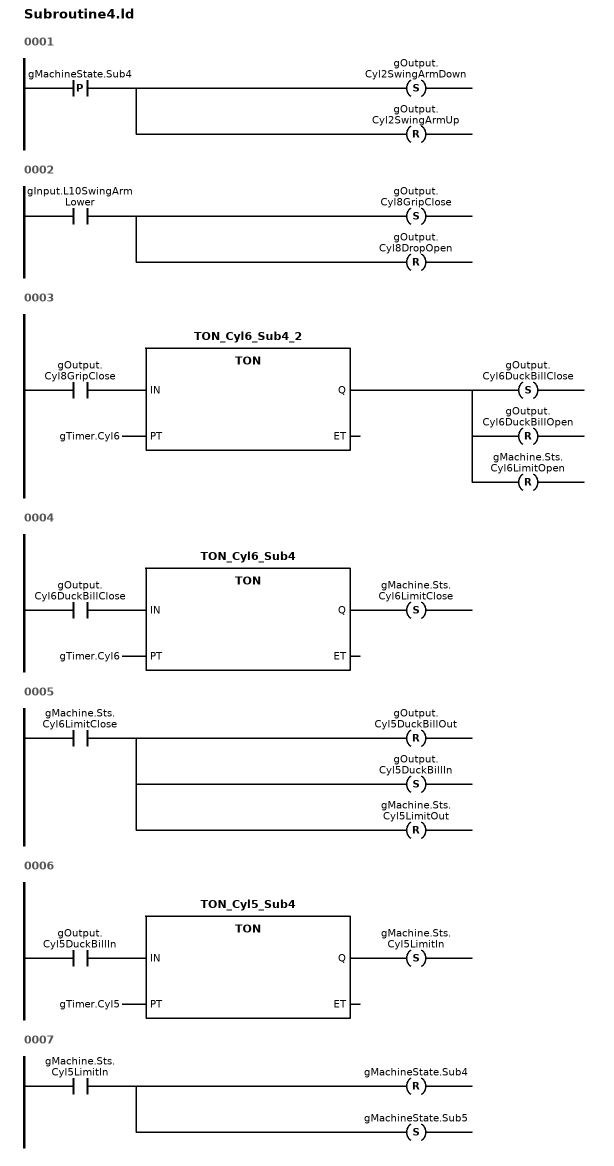
Ladder, written as Structured Text:
```iecst
ACTION Subroutine4:
VAR
    _e1 : R_TRIG;
END_VAR
(* Network 1 *)
_e1(CLK := gMachineState.Sub4);
IF _e1.Q THEN
    gOutput.Cyl2SwingArmDown := TRUE;
    gOutput.Cyl2SwingArmUp := FALSE;
END_IF;

(* Network 2 *)
IF gInput.L10SwingArmLower THEN
    gOutput.Cyl8GripClose := TRUE;
    gOutput.Cyl8DropOpen := FALSE;
END_IF;

(* Network 3 *)
TON_Cyl6_Sub4_2(IN := gOutput.Cyl8GripClose, PT := gTimer.Cyl6);
IF TON_Cyl6_Sub4_2.Q THEN
    gOutput.Cyl6DuckBillClose := TRUE;
    gOutput.Cyl6DuckBillOpen := FALSE;
    gMachine.Sts.Cyl6LimitOpen := FALSE;
END_IF;

(* Network 4 *)
TON_Cyl6_Sub4(IN := gOutput.Cyl6DuckBillClose, PT := gTimer.Cyl6);
IF TON_Cyl6_Sub4.Q THEN gMachine.Sts.Cyl6LimitClose := TRUE; END_IF;

(* Network 5 *)
IF gMachine.Sts.Cyl6LimitClose THEN
    gOutput.Cyl5DuckBillOut := FALSE;
    gOutput.Cyl5DuckBillIn := TRUE;
    gMachine.Sts.Cyl5LimitOut := FALSE;
END_IF;

(* Network 6 *)
TON_Cyl5_Sub4(IN := gOutput.Cyl5DuckBillIn, PT := gTimer.Cyl5);
IF TON_Cyl5_Sub4.Q THEN gMachine.Sts.Cyl5LimitIn := TRUE; END_IF;

(* Network 7 *)
IF gMachine.Sts.Cyl5LimitIn THEN
    gMachineState.Sub4 := FALSE;
    gMachineState.Sub5 := TRUE;
END_IF;
END_ACTION
```

#### Subroutine5.ld - Swing upwards with bag
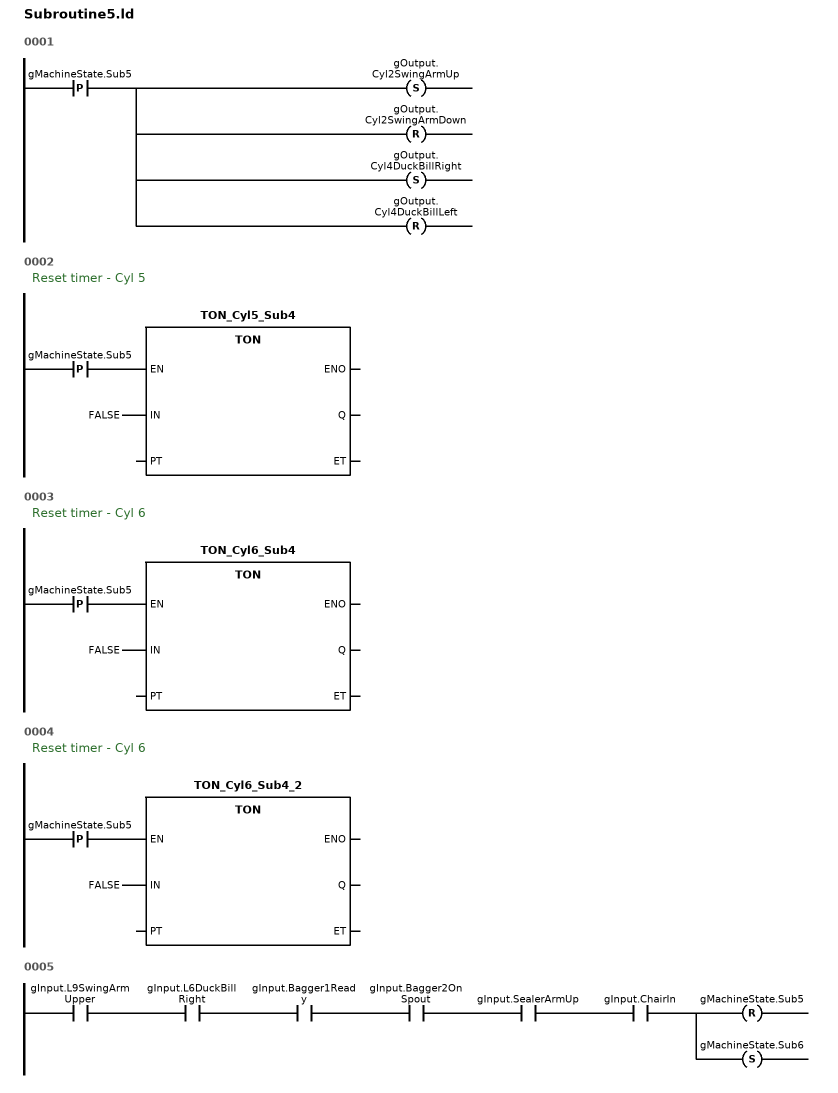
Ladder, written as Structured Text:
```iecst
ACTION Subroutine5:
VAR
    _e1 : R_TRIG;
    _e2 : R_TRIG;
    _e3 : R_TRIG;
    _e4 : R_TRIG;
    _p5 : BOOL;
END_VAR
(* Network 1 *)
_e1(CLK := gMachineState.Sub5);
IF _e1.Q THEN
    gOutput.Cyl2SwingArmUp := TRUE;
    gOutput.Cyl2SwingArmDown := FALSE;
    gOutput.Cyl4DuckBillRight := TRUE;
    gOutput.Cyl4DuckBillLeft := FALSE;
END_IF;

(* Network 2: Reset timer - Cyl 5 *)
_e2(CLK := gMachineState.Sub5);
IF _e2.Q THEN TON_Cyl5_Sub4(IN := FALSE); END_IF;

(* Network 3: Reset timer - Cyl 6 *)
_e3(CLK := gMachineState.Sub5);
IF _e3.Q THEN TON_Cyl6_Sub4(IN := FALSE); END_IF;

(* Network 4: Reset timer - Cyl 6 *)
_e4(CLK := gMachineState.Sub5);
IF _e4.Q THEN TON_Cyl6_Sub4_2(IN := FALSE); END_IF;

(* Network 5 *)
_p5 := gInput.L9SwingArmUpper AND gInput.L6DuckBillRight AND gInput.Bagger1Ready AND gInput.Bagger2OnSpout AND gInput.SealerArmUp AND gInput.ChairIn;
IF _p5 THEN
    gMachineState.Sub5 := FALSE;
    gMachineState.Sub6 := TRUE;
END_IF;
END_ACTION
```

#### Subroutine6.ld - Move carriage to bag filling machine
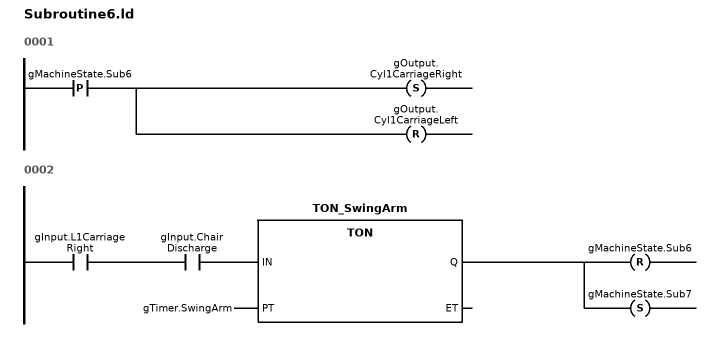
Ladder, written as Structured Text:
```iecst
ACTION Subroutine6:
VAR
    _e1 : R_TRIG;
END_VAR
(* Network 1 *)
_e1(CLK := gMachineState.Sub6);
IF _e1.Q THEN
    gOutput.Cyl1CarriageRight := TRUE;
    gOutput.Cyl1CarriageLeft := FALSE;
END_IF;

(* Network 2 *)
TON_SwingArm(IN := gInput.L1CarriageRight AND gInput.ChairDischarge, PT := gTimer.SwingArm);
IF TON_SwingArm.Q THEN
    gMachineState.Sub6 := FALSE;
    gMachineState.Sub7 := TRUE;
END_IF;
END_ACTION
```

#### Subroutine7.ld - Swing bag onto bag filling spout
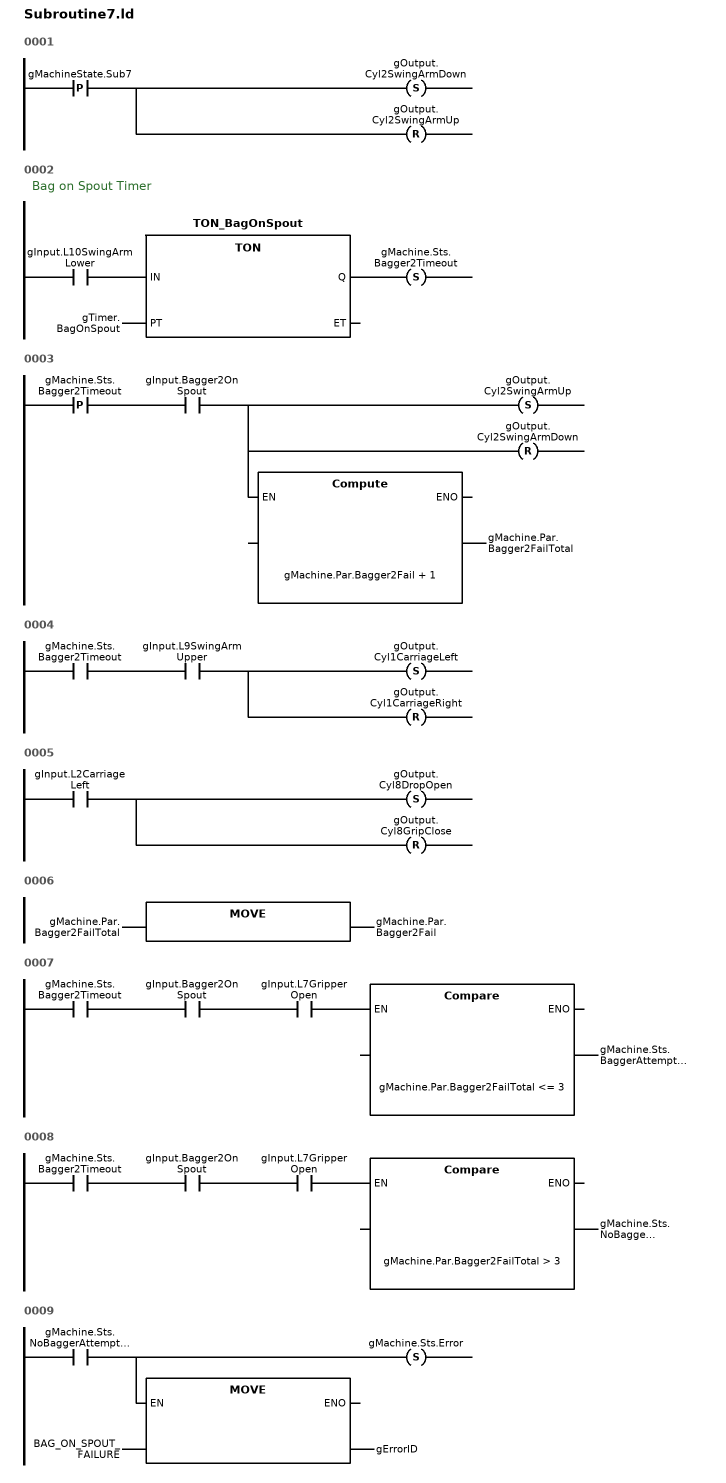
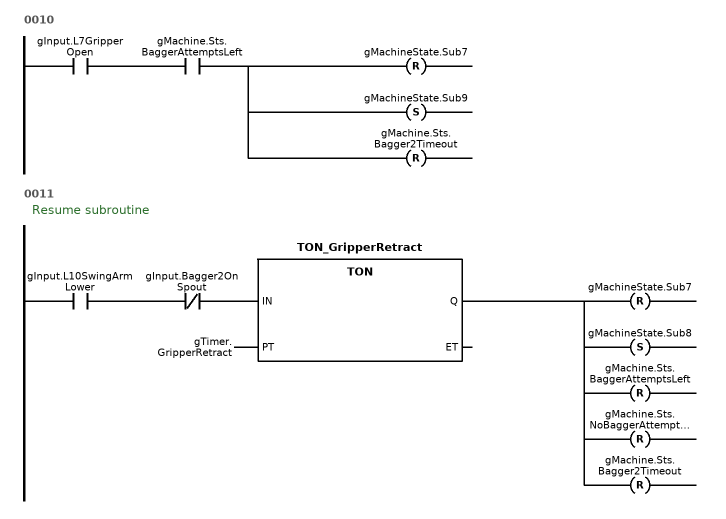
Ladder, written as Structured Text:
```iecst
ACTION Subroutine7:
VAR
    _e1 : R_TRIG;
    _e2 : R_TRIG;
    _p3 : BOOL;
    _p4 : BOOL;
    _p5 : BOOL;
    _p6 : BOOL;
    _p7 : BOOL;
END_VAR
(* Network 1 *)
_e1(CLK := gMachineState.Sub7);
IF _e1.Q THEN
    gOutput.Cyl2SwingArmDown := TRUE;
    gOutput.Cyl2SwingArmUp := FALSE;
END_IF;

(* Network 2: Bag on Spout Timer *)
TON_BagOnSpout(IN := gInput.L10SwingArmLower, PT := gTimer.BagOnSpout);
IF TON_BagOnSpout.Q THEN gMachine.Sts.Bagger2Timeout := TRUE; END_IF;

(* Network 3 *)
_e2(CLK := gMachine.Sts.Bagger2Timeout);
IF _e2.Q AND gInput.Bagger2OnSpout THEN
    gOutput.Cyl2SwingArmUp := TRUE;
    gOutput.Cyl2SwingArmDown := FALSE;
    gMachine.Par.Bagger2FailTotal := gMachine.Par.Bagger2Fail + 1;
END_IF;

(* Network 4 *)
_p3 := gMachine.Sts.Bagger2Timeout AND gInput.L9SwingArmUpper;
IF _p3 THEN
    gOutput.Cyl1CarriageLeft := TRUE;
    gOutput.Cyl1CarriageRight := FALSE;
END_IF;

(* Network 5 *)
IF gInput.L2CarriageLeft THEN
    gOutput.Cyl8DropOpen := TRUE;
    gOutput.Cyl8GripClose := FALSE;
END_IF;

(* Network 6 *)
gMachine.Par.Bagger2Fail := gMachine.Par.Bagger2FailTotal;

(* Network 7 *)
_p4 := gMachine.Sts.Bagger2Timeout AND gInput.Bagger2OnSpout AND gInput.L7GripperOpen;
IF _p4 THEN gMachine.Sts.BaggerAttemptsLeft := gMachine.Par.Bagger2FailTotal <= 3; END_IF;

(* Network 8 *)
_p5 := gMachine.Sts.Bagger2Timeout AND gInput.Bagger2OnSpout AND gInput.L7GripperOpen;
IF _p5 THEN gMachine.Sts.NoBaggerAttemptsLeft := gMachine.Par.Bagger2FailTotal > 3; END_IF;

(* Network 9 *)
_p6 := gMachine.Sts.NoBaggerAttemptsLeft;
IF gMachine.Sts.NoBaggerAttemptsLeft THEN gMachine.Sts.Error := TRUE; END_IF;
IF _p6 THEN gErrorID := BAG_ON_SPOUT_FAILURE; END_IF;

(* Network 10 *)
_p7 := gInput.L7GripperOpen AND gMachine.Sts.BaggerAttemptsLeft;
IF _p7 THEN
    gMachineState.Sub7 := FALSE;
    gMachineState.Sub9 := TRUE;
    gMachine.Sts.Bagger2Timeout := FALSE;
END_IF;

(* Network 11: Resume subroutine *)
TON_GripperRetract(IN := gInput.L10SwingArmLower AND NOT gInput.Bagger2OnSpout, PT := gTimer.GripperRetract);
IF TON_GripperRetract.Q THEN
    gMachineState.Sub7 := FALSE;
    gMachineState.Sub8 := TRUE;
    gMachine.Sts.BaggerAttemptsLeft := FALSE;
    gMachine.Sts.NoBaggerAttemptsLeft := FALSE;
    gMachine.Sts.Bagger2Timeout := FALSE;
END_IF;
END_ACTION
```

#### Subroutine8.ld - Release bag
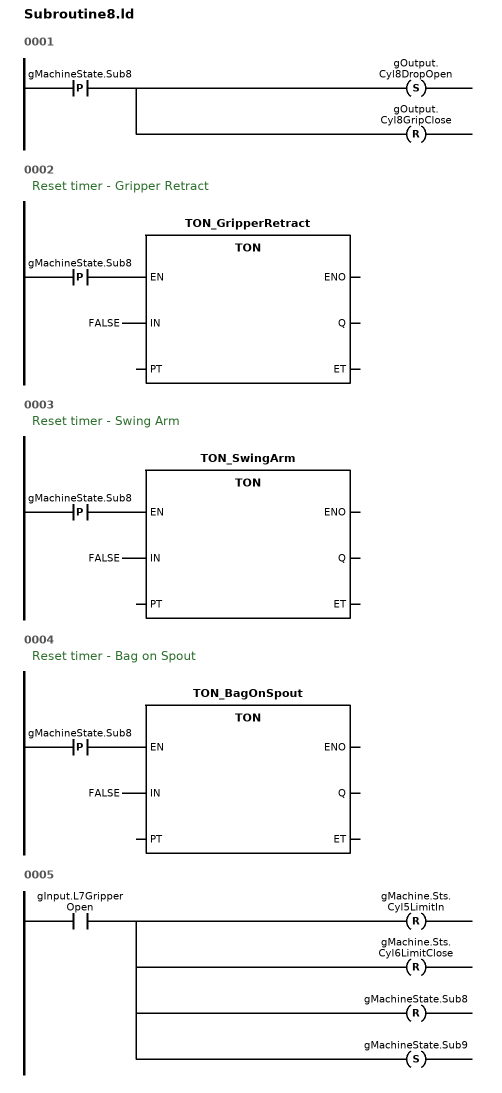
Ladder, written as Structured Text:
```iecst
ACTION Subroutine8:
VAR
    _e1 : R_TRIG;
    _e2 : R_TRIG;
    _e3 : R_TRIG;
    _e4 : R_TRIG;
END_VAR
(* Network 1 *)
_e1(CLK := gMachineState.Sub8);
IF _e1.Q THEN
    gOutput.Cyl8DropOpen := TRUE;
    gOutput.Cyl8GripClose := FALSE;
END_IF;

(* Network 2: Reset timer - Gripper Retract *)
_e2(CLK := gMachineState.Sub8);
IF _e2.Q THEN TON_GripperRetract(IN := FALSE); END_IF;

(* Network 3: Reset timer - Swing Arm *)
_e3(CLK := gMachineState.Sub8);
IF _e3.Q THEN TON_SwingArm(IN := FALSE); END_IF;

(* Network 4: Reset timer - Bag on Spout *)
_e4(CLK := gMachineState.Sub8);
IF _e4.Q THEN TON_BagOnSpout(IN := FALSE); END_IF;

(* Network 5 *)
IF gInput.L7GripperOpen THEN
    gMachine.Sts.Cyl5LimitIn := FALSE;
    gMachine.Sts.Cyl6LimitClose := FALSE;
    gMachineState.Sub8 := FALSE;
    gMachineState.Sub9 := TRUE;
END_IF;
END_ACTION
```

#### Subroutine9.ld - Repeat
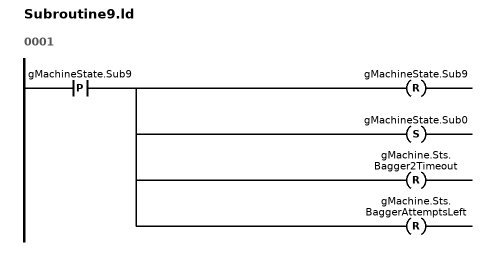
Ladder, written as Structured Text:
```iecst
ACTION Subroutine9:
VAR
    _e1 : R_TRIG;
END_VAR
(* Network 1 *)
_e1(CLK := gMachineState.Sub9);
IF _e1.Q THEN
    gMachineState.Sub9 := FALSE;
    gMachineState.Sub0 := TRUE;
    gMachine.Sts.Bagger2Timeout := FALSE;
    gMachine.Sts.BaggerAttemptsLeft := FALSE;
END_IF;
END_ACTION
```

#### CheckError.ld -  Error handling
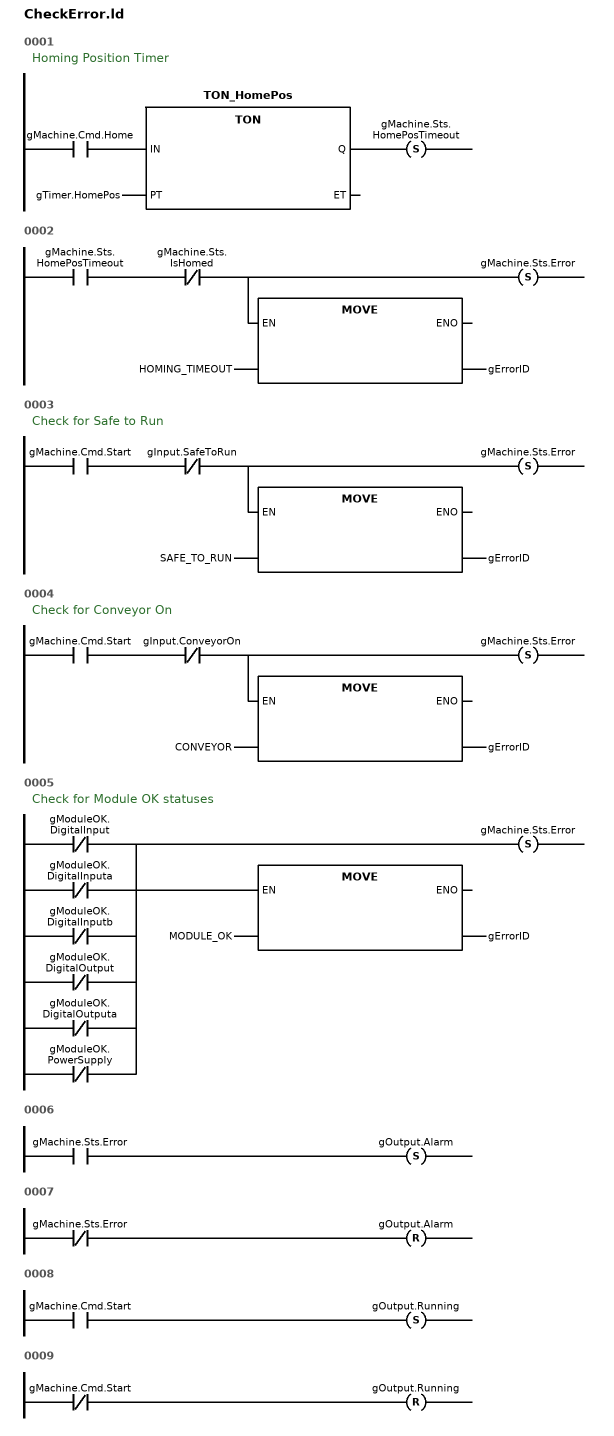
Ladder, written as Structured Text:
```iecst
ACTION CheckError:
VAR
    _p1 : BOOL;
    _p2 : BOOL;
    _p3 : BOOL;
END_VAR
(* Network 1: Homing Position Timer *)
TON_HomePos(IN := gMachine.Cmd.Home, PT := gTimer.HomePos);
IF TON_HomePos.Q THEN gMachine.Sts.HomePosTimeout := TRUE; END_IF;

(* Network 2 *)
_p1 := gMachine.Sts.HomePosTimeout AND NOT gMachine.Sts.IsHomed;
IF _p1 THEN
    gMachine.Sts.Error := TRUE;
    gErrorID := HOMING_TIMEOUT;
END_IF;

(* Network 3: Check for Safe to Run *)
_p2 := gMachine.Cmd.Start AND NOT gInput.SafeToRun;
IF gMachine.Cmd.Start AND NOT gInput.SafeToRun THEN gMachine.Sts.Error := TRUE; END_IF;
IF _p2 THEN gErrorID := SAFE_TO_RUN; END_IF;

(* Network 4: Check for Conveyor On *)
_p3 := gMachine.Cmd.Start AND NOT gInput.ConveyorOn;
IF gMachine.Cmd.Start AND NOT gInput.ConveyorOn THEN gMachine.Sts.Error := TRUE; END_IF;
IF _p3 THEN gErrorID := CONVEYOR; END_IF;

(* Network 5: Check for Module OK statuses *)
IF NOT gModuleOK.DigitalInput OR NOT gModuleOK.DigitalInputa OR NOT gModuleOK.DigitalInputb OR NOT gModuleOK.DigitalOutput OR NOT gModuleOK.DigitalOutputa OR NOT gModuleOK.PowerSupply THEN
    gMachine.Sts.Error := TRUE;
    gErrorID := MODULE_OK;
END_IF;

(* Network 6 *)
IF gMachine.Sts.Error THEN gOutput.Alarm := TRUE; END_IF;

(* Network 7 *)
IF NOT gMachine.Sts.Error THEN gOutput.Alarm := FALSE; END_IF;

(* Network 8 *)
IF gMachine.Cmd.Start THEN gOutput.Running := TRUE; END_IF;

(* Network 9 *)
IF NOT gMachine.Cmd.Start THEN gOutput.Running := FALSE; END_IF;
END_ACTION
```

#### Stop.ld - Stop machine
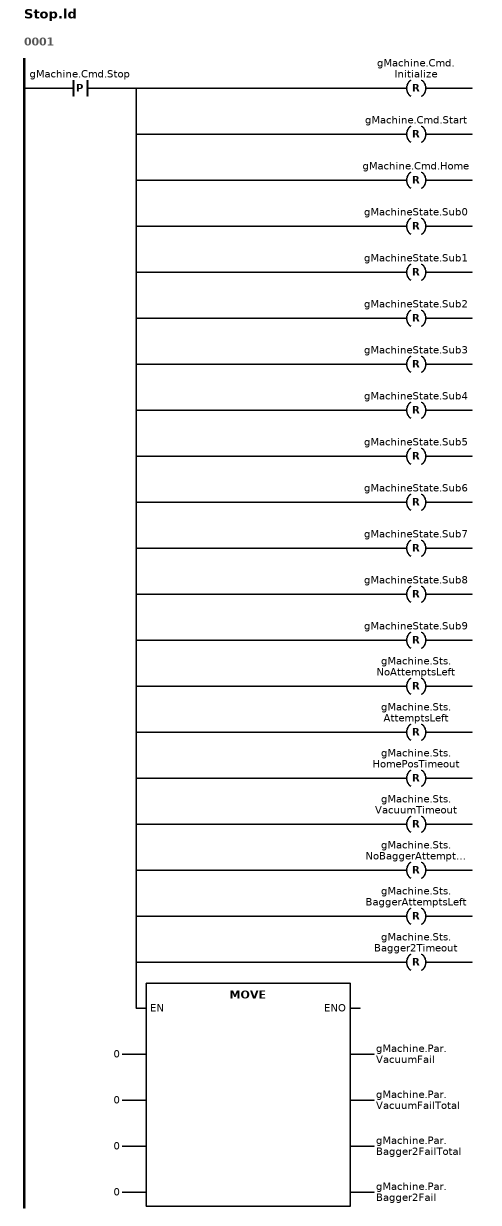
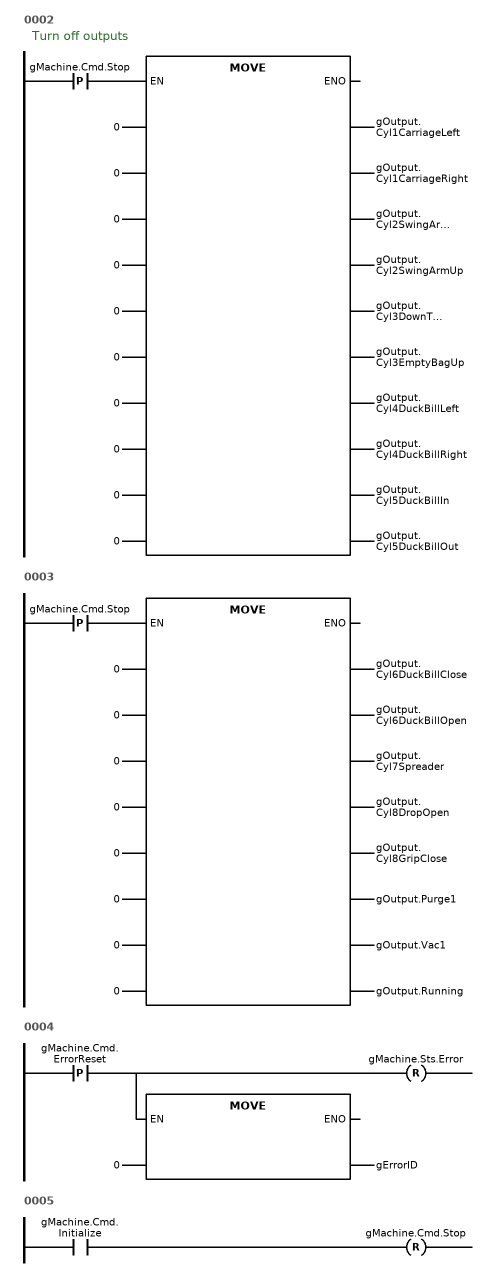
Ladder, written as Structured Text:
```iecst
ACTION Stop:
VAR
    _e1 : R_TRIG;
    _e2 : R_TRIG;
    _e3 : R_TRIG;
    _e4 : R_TRIG;
END_VAR
(* Network 1 *)
_e1(CLK := gMachine.Cmd.Stop);
IF _e1.Q THEN
    gMachine.Cmd.Initialize := FALSE;
    gMachine.Cmd.Start := FALSE;
    gMachine.Cmd.Home := FALSE;
    gMachineState.Sub0 := FALSE;
    gMachineState.Sub1 := FALSE;
    gMachineState.Sub2 := FALSE;
    gMachineState.Sub3 := FALSE;
    gMachineState.Sub4 := FALSE;
    gMachineState.Sub5 := FALSE;
    gMachineState.Sub6 := FALSE;
    gMachineState.Sub7 := FALSE;
    gMachineState.Sub8 := FALSE;
    gMachineState.Sub9 := FALSE;
    gMachine.Sts.NoAttemptsLeft := FALSE;
    gMachine.Sts.AttemptsLeft := FALSE;
    gMachine.Sts.HomePosTimeout := FALSE;
    gMachine.Sts.VacuumTimeout := FALSE;
    gMachine.Sts.NoBaggerAttemptsLeft := FALSE;
    gMachine.Sts.BaggerAttemptsLeft := FALSE;
    gMachine.Sts.Bagger2Timeout := FALSE;
    gMachine.Par.VacuumFail := 0;
    gMachine.Par.VacuumFailTotal := 0;
    gMachine.Par.Bagger2FailTotal := 0;
    gMachine.Par.Bagger2Fail := 0;
END_IF;

(* Network 2: Turn off outputs *)
_e2(CLK := gMachine.Cmd.Stop);
IF _e2.Q THEN
    gOutput.Cyl1CarriageLeft := 0;
    gOutput.Cyl1CarriageRight := 0;
    gOutput.Cyl2SwingArmDown := 0;
    gOutput.Cyl2SwingArmUp := 0;
    gOutput.Cyl3DownToEmptyBag := 0;
    gOutput.Cyl3EmptyBagUp := 0;
    gOutput.Cyl4DuckBillLeft := 0;
    gOutput.Cyl4DuckBillRight := 0;
    gOutput.Cyl5DuckBillIn := 0;
    gOutput.Cyl5DuckBillOut := 0;
END_IF;

(* Network 3 *)
_e3(CLK := gMachine.Cmd.Stop);
IF _e3.Q THEN
    gOutput.Cyl6DuckBillClose := 0;
    gOutput.Cyl6DuckBillOpen := 0;
    gOutput.Cyl7Spreader := 0;
    gOutput.Cyl8DropOpen := 0;
    gOutput.Cyl8GripClose := 0;
    gOutput.Purge1 := 0;
    gOutput.Vac1 := 0;
    gOutput.Running := 0;
END_IF;

(* Network 4 *)
_e4(CLK := gMachine.Cmd.ErrorReset);
IF _e4.Q THEN
    gMachine.Sts.Error := FALSE;
    gErrorID := 0;
END_IF;

(* Network 5 *)
IF gMachine.Cmd.Initialize THEN gMachine.Cmd.Stop := FALSE; END_IF;
END_ACTION
```
